FUNCTION_BLOCK SimplePositionBehaviour IMPLEMENTS I_Task
VAR_INPUT
END_VAR
VAR_OUTPUT
END_VAR
VAR
	moveAbs	: MC_MoveAbsolute;
	_Axis : REFERENCE TO AXIS_REF;
	MoveToPos : BOOL;
	State: INT;
	_Done: BOOL;
	_Error: BOOL;
	_Busy: BOOL;
END_VAR

{analysis -2}

METHOD Abort : BOOL
moveAbs.Execute := FALSE;
moveAbs.Position := moveAbs.Velocity := 0;
MoveToPos := false;
_Busy := false;
Abort := true;
State := 0;
END_METHOD

PROPERTY PUBLIC Acceleration : mc_lreal
GET
Acceleration := moveAbs.Acceleration;
END_GET
SET
moveAbs.Acceleration := Acceleration;
END_SET
END_PROPERTY

PROPERTY Busy : BOOL
GET
Busy := _Busy;
END_GET
END_PROPERTY

METHOD Cycle : HRESULT
VAR_INPUT
END_VAR
Cycle := S_OK;
CASE State OF
	0:
		IF moveAbs.Busy THEN
			State := 10;
			MoveToPos := FALSE;
		END_IF
	
	10:
		IF NOT moveAbs.Busy THEN
			IF moveAbs.Done THEN
				_Done := TRUE;
			ELSIF moveAbs.Error THEN
				_Error := TRUE;
			END_IF
			_Busy := FALSE;
			moveAbs.Execute := FALSE;
			State := 0;
			Cycle := S_OK;
		END_IF
	ELSE
		Cycle := E_FAIL;
END_CASE

moveAbs(Axis := _Axis);
END_METHOD

PROPERTY PUBLIC Deceleration : mc_lreal
GET
Deceleration := moveAbs.Deceleration;
END_GET
SET
moveAbs.Deceleration := Deceleration;
END_SET
END_PROPERTY

PROPERTY Done : BOOL
GET
Done := _Done;
END_GET
END_PROPERTY

PROPERTY Error : BOOL
GET
Error := _Error;
END_GET
END_PROPERTY

METHOD FB_init : BOOL
VAR_INPUT
	bInitRetains : BOOL; // if TRUE, the retain variables are initialized (warm start / cold start)
	bInCopyCode : BOOL;  // if TRUE, the instance afterwards gets moved into the copy code (online change)
	axis : reference TO AXIS_REF;
END_VAR
_Axis REF= axis;
END_METHOD

PROPERTY PUBLIC Jerk : mc_lreal
GET
Jerk := moveAbs.Jerk;
END_GET
SET
moveAbs.Jerk := Jerk;
END_SET
END_PROPERTY

METHOD MoveTo : BOOL
VAR_INPUT
	Position : MC_LREAL;
	Velocity : MC_LREAL;
	Task : REFERENCE TO I_Task;
END_VAR
moveAbs.Position := Position;
moveAbs.Velocity := Velocity;
MoveTo := TRUE;
Task := THIS^;
_Done := FALSE;
_Error := FALSE;
_Busy := TRUE;
moveAbs.Execute := TRUE;
END_METHOD

END_FUNCTION_BLOCK

(* stored: Version 1.1.0.1
   POU SimplePositionBehaviour: Id {28fa9c58-d811-4345-8e27-94422602642f}, SpecialFunc None
   Method Abort: Id {1cd0d7f2-688c-4d35-83e4-94847f46cad7}
   Property Acceleration: Id {3af53338-23b7-44e8-b1be-bfde3ab4639f}
   Get Get: Id {6ee0cb9a-1db1-4f3d-bd00-5f31376a507f}
   Set Set: Id {9065b1b0-2b4a-4502-a521-32f63bb5796b}
   Property Busy: Id {15fd35de-807b-4d13-84bf-f7daa15c531a}
   Get Get: Id {052fd6fa-89c7-4920-8bdf-0578104cda0f}
   Method Cycle: Id {a39af4f2-815a-48ca-8486-fcba13c88617}
   Property Deceleration: Id {207379d4-5297-4661-a6b0-70afa1cf5253}
   Get Get: Id {2b3ec42b-d81e-4e4f-a5e5-4d4d8d1cc1cd}
   Set Set: Id {c421d552-e5af-44da-9f19-63ad72f26836}
   Property Done: Id {03fb8255-039b-454a-b329-0c2121d24eb2}
   Get Get: Id {98bc89bd-bc6c-43b4-aec6-075eea67c7b3}
   Property Error: Id {780892dd-fd19-47af-926f-a732f401392e}
   Get Get: Id {b0c83e66-5dc8-4591-bc9b-cf6a1c94a587}
   Method FB_init: Id {0156f89a-4ccc-4fea-9390-c950d3f5d691}
   Property Jerk: Id {ad403219-1be7-4bab-be70-39ef22f28e38}
   Get Get: Id {d61d7606-d3eb-410b-8474-a2e97b22b31e}
   Set Set: Id {ecb0ed4b-5217-48bc-9bfd-1f75c1a8109f}
   Method MoveTo: Id {a8cef16b-0fac-4b3b-9508-699ac7e78071} *)
